// SIMATIC S7-200 project (STEP 7-Micro/WIN), CPU 221 REL 01.10

SYMBOL_TABLE USR1
Always_On        SM0.0    // This bit is always on.
Hours            VW0      // Stores the measured number of hours the device has been operating.
Minutes          VW2      // Stores the measured number of minutes the device has been operating.
Seconds          VW4      // Stores the measured number of seconds the device has been operating.
Output_LEDs      QB0      // LEDs for displaying number of seconds the device has been operational.
END_SYMBOL_TABLE

ORGANIZATION_BLOCK MAIN:OB1
TITLE=
//  题目：怎样追踪一台设备运行了多长时间
//  ***概述***
// 本例程序的目的是纪录一台设备（制动器、开关等）运行的时间，以下前提必须
// 满足：当设备运行时，必须给输入I0.0提供24V信号；当设备不工作时不提供电压。
// 当提供输入信号时，开始测量时间。如果没有输入信号，那么就中断时间的测量，
// 直到重新提供输入信号为止。测量到的小时数存在字VWD中，分钟数存在字VW2中，
// 秒数存在VW4中。
// ***程序和注释***
// 程序第一个扫描周期调用子程序1。在子程序1中，设定计时器T5为1秒的运行时间，
// 当达到1秒时，计时器位“T5"被置1，同时秒计数标志VW4增加1，并将计时器位“T5"复位
// 因此，计时器能在下一周期立即重新起动。
// 当秒计数标志达到60时，分钟计数标志VW2加1，秒计数标志VW4被置为0。
// 当分计数标志达到60时，小时计数标志VW0加1，分钟计数标志VW2被置为0。子程序结束。
// 主程序结束的最后一行用二进制来显示当前的秒数，用输出端的LED显示。
// 标题：计时器
// 
BEGIN
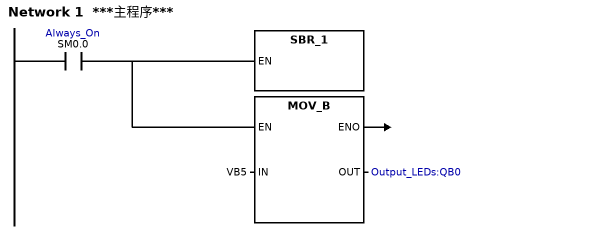
Network 1 // ***主程序***
// SM0.0总是1
// 调用测量子程序1
// 在输出QB0的LED上显示秒数
LD     Always_On:SM0.0
CALL   SBR_1:SBR1
MOVB   VB5, Output_LEDs:QB0
Network 2 // 主程序结束
// MEND
// 
Network 3 // ***子程序1***
END_ORGANIZATION_BLOCK

SUBROUTINE_BLOCK SBR_1:SBR1
TITLE=
BEGIN
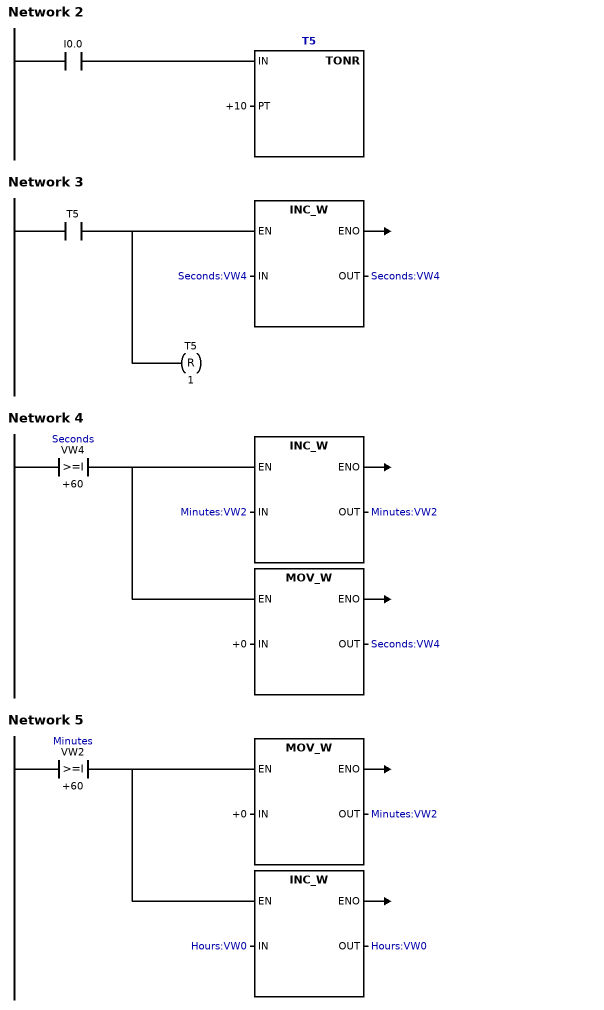
Network 2
// 测量输入I0.0的运行时间。如果I0.0=1,则
// 设定计时器时间为1s
LD     I0.0
TONR   T5, +10
Network 3
// 如果达到1秒
// 则秒计数器加1
// 秒计数器复位
LD     T5
INCW   Seconds:VW4
R      T5, 1
Network 4
// 若计数到60秒					// If VW4>=60,
// 则分寄存器加1
// 秒寄存器清零
LDW>=  Seconds:VW4, +60
INCW   Minutes:VW2
MOVW   +0, Seconds:VW4
Network 5
// 若计数到60分
//分计数标志清零
//时计数标志加1
LDW>=  Minutes:VW2, +60
MOVW   +0, Minutes:VW2
INCW   Hours:VW0
Network 6 //  测量子程序结束
// RET				
// 
END_SUBROUTINE_BLOCK
